FUNCTION_BLOCK AX_SEL_BYTE (* binary selection *)
  (* Standard: 61131-3; Classification: standard selection function; Description: Copyright (c) 2012 TU Wien ACIN, HR Agrartechnik GmbH This program and the accompanying materials are made available under the terms of the Eclipse Public License 2.0 which is available at https://www.eclipse.org/legal/epl-2.0/ SPDX-License-Identifier: EPL-2.0 *)
  (* Version 3.1, 2026-07-04, Franz Höpfinger, HR Agrartechnik GmbH, added note: an output event is only generated if G changes! *)
  (* Version 3.0, 2025-04-14, Patrick Aigner, changed package *)
  (* Version 1.0, 2012-03-25, Monika Wenger, TU Wien ACIN, initial API and implementation and/or initial documentation *)
  PACKAGE adapter::iec61131::selection;
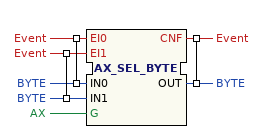
  EVENT_INPUT
    EI0 WITH IN0; (* Set IN0 *)
    EI1 WITH IN1; (* Set IN1 *)
  END_EVENT
  EVENT_OUTPUT
    CNF WITH OUT; (* Confirmation of Requested Service *)
  END_EVENT
  VAR_INPUT
    IN0 : BYTE; (* Selectable input variable *)
    IN1 : BYTE; (* Selectable input variable *)
  END_VAR
  VAR_OUTPUT
    OUT : BYTE; (* Selected input *)
  END_VAR
  SOCKETS
    G : adapter::types::unidirectional::AX; (* Selelctor *)
  END_SOCKETS
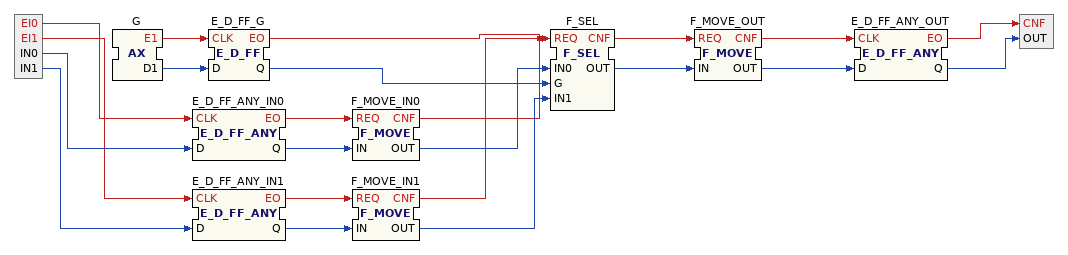
  FBS
    F_MOVE_IN1 : iec61131::selection::F_MOVE; {SET_ATTRIBUTE(DataType, BYTE)}
    E_D_FF_ANY_IN0 : iec61499::events::E_D_FF_ANY;
    F_MOVE_IN0 : iec61131::selection::F_MOVE; {SET_ATTRIBUTE(DataType, BYTE)}
    E_D_FF_G : iec61499::events::E_D_FF;
    E_D_FF_ANY_IN1 : iec61499::events::E_D_FF_ANY;
    E_D_FF_ANY_OUT : iec61499::events::E_D_FF_ANY;
    F_SEL : iec61131::selection::F_SEL;
    F_MOVE_OUT : iec61131::selection::F_MOVE; {SET_ATTRIBUTE(DataType, BYTE)}
  END_FBS
  EVENT_CONNECTIONS
    F_SEL.CNF TO F_MOVE_OUT.REQ;
    E_D_FF_ANY_IN1.EO TO F_MOVE_IN1.REQ;
    F_MOVE_IN1.CNF TO F_SEL.REQ;
    F_MOVE_IN0.CNF TO F_SEL.REQ;
    F_MOVE_OUT.CNF TO E_D_FF_ANY_OUT.CLK;
    E_D_FF_ANY_IN0.EO TO F_MOVE_IN0.REQ;
    E_D_FF_G.EO TO F_SEL.REQ;
    G.E1 TO E_D_FF_G.CLK;
    EI1 TO E_D_FF_ANY_IN1.CLK;
    EI0 TO E_D_FF_ANY_IN0.CLK;
    E_D_FF_ANY_OUT.EO TO CNF;
  END_CONNECTIONS
  DATA_CONNECTIONS
    E_D_FF_ANY_IN1.Q TO F_MOVE_IN1.IN;
    E_D_FF_ANY_IN0.Q TO F_MOVE_IN0.IN;
    F_MOVE_IN0.OUT TO F_SEL.IN0;
    E_D_FF_G.Q TO F_SEL.G;
    F_SEL.OUT TO F_MOVE_OUT.IN;
    F_MOVE_OUT.OUT TO E_D_FF_ANY_OUT.D;
    F_MOVE_IN1.OUT TO F_SEL.IN1;
    G.D1 TO E_D_FF_G.D;
    IN1 TO E_D_FF_ANY_IN1.D;
    IN0 TO E_D_FF_ANY_IN0.D;
    E_D_FF_ANY_OUT.Q TO OUT;
  END_CONNECTIONS
END_FUNCTION_BLOCK
